ABB RAPID module: 0016EFE6

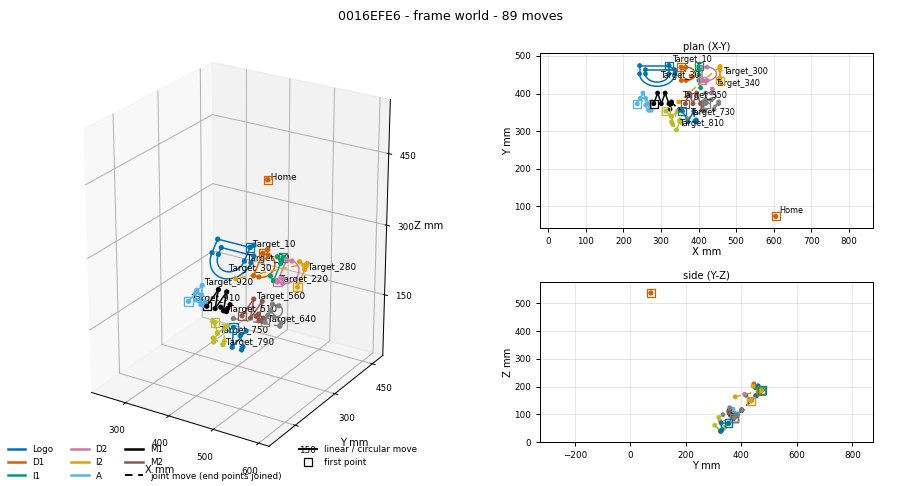
[picture p0: tool path of 0016EFE6 in frame world, 89 of 89 moves have a stored position in this frame; points joined in program order, loops and branches not executed]
MODULE Module1
    CONST robtarget Target_360:=[[614.368006487,-305.026841829,-535.49276156],[0.482962895,-0.129409515,-0.299950184,0.812422247],[-1,0,0,0],[9E+09,9E+09,9E+09,9E+09,9E+09,9E+09]];
    CONST robtarget Target_370:=[[614.368006487,-305.026841829,-535.49276156],[0.482962895,-0.129409515,-0.299950184,0.812422247],[-1,0,0,0],[9E+09,9E+09,9E+09,9E+09,9E+09,9E+09]];
    CONST robtarget Target_380:=[[614.368006487,-305.026841829,-535.49276156],[0.482962895,-0.129409515,-0.299950184,0.812422247],[-1,0,0,0],[9E+09,9E+09,9E+09,9E+09,9E+09,9E+09]];
    CONST robtarget Target_410:=[[614.368006487,-305.026841829,-535.49276156],[0.482962895,-0.129409515,-0.299950184,0.812422247],[-1,0,0,0],[9E+09,9E+09,9E+09,9E+09,9E+09,9E+09]];
    CONST robtarget Target_390:=[[614.368006487,-305.026841829,-535.49276156],[0.482962895,-0.129409515,-0.299950184,0.812422247],[-1,0,0,0],[9E+09,9E+09,9E+09,9E+09,9E+09,9E+09]];
    CONST robtarget Target_400:=[[614.368006487,-305.026841829,-535.49276156],[0.482962895,-0.129409515,-0.299950184,0.812422247],[-1,0,0,0],[9E+09,9E+09,9E+09,9E+09,9E+09,9E+09]];
    CONST robtarget Target_420:=[[614.368006487,-305.026841829,-535.49276156],[0.482962895,-0.129409515,-0.299950184,0.812422247],[-1,0,0,0],[9E+09,9E+09,9E+09,9E+09,9E+09,9E+09]];
    CONST robtarget Target_430:=[[614.368006487,-305.026841829,-535.49276156],[0.482962895,-0.129409515,-0.299950184,0.812422247],[-1,0,0,0],[9E+09,9E+09,9E+09,9E+09,9E+09,9E+09]];
    CONST robtarget Target_440:=[[614.368006487,-305.026841829,-535.49276156],[0.482962895,-0.129409515,-0.299950184,0.812422247],[-1,0,0,0],[9E+09,9E+09,9E+09,9E+09,9E+09,9E+09]];
    CONST robtarget Target_450:=[[614.368006487,-305.026841829,-535.49276156],[0.482962895,-0.129409515,-0.299950184,0.812422247],[-1,0,0,0],[9E+09,9E+09,9E+09,9E+09,9E+09,9E+09]];
    CONST robtarget Target_550:=[[186.614,135,0],[1,0,0,0],[0,0,0,0],[9E+09,9E+09,9E+09,9E+09,9E+09,9E+09]];
    CONST robtarget Target_560:=[[146.614,125,0],[1,0,0,0],[0,-2,1,0],[9E+09,9E+09,9E+09,9E+09,9E+09,9E+09]];
    CONST robtarget Target_570:=[[186.614,115,0],[1,0,0,0],[0,-2,1,0],[9E+09,9E+09,9E+09,9E+09,9E+09,9E+09]];
    CONST robtarget Target_580:=[[146.614,105,0],[1,0,0,0],[0,-2,1,0],[9E+09,9E+09,9E+09,9E+09,9E+09,9E+09]];
    CONST robtarget Target_590:=[[186.614,95,0],[1,0,0,0],[0,-2,1,0],[9E+09,9E+09,9E+09,9E+09,9E+09,9E+09]];
    CONST robtarget Target_620:=[[186.614143087,91.364778393,-24.569544894],[1,-0.00000011,0.000000243,0.000000801],[0,-2,1,0],[9E+09,9E+09,9E+09,9E+09,9E+09,9E+09]];
    CONST robtarget Target_600:=[[186.614,88,0],[1,0,0,0],[0,-2,1,0],[9E+09,9E+09,9E+09,9E+09,9E+09,9E+09]];
    CONST robtarget Target_610:=[[179.614,88,0],[1,0,0,0],[0,-2,1,0],[9E+09,9E+09,9E+09,9E+09,9E+09,9E+09]];
    CONST robtarget Target_630:=[[182.856287812,84.770817951,-30.544070021],[1,0.000000024,0.000000045,0.000000006],[0,-2,1,0],[9E+09,9E+09,9E+09,9E+09,9E+09,9E+09]];
    CONST robtarget Target_10:=[[43.067,178.883,0],[1,0,0,0],[0,-2,1,0],[9E+09,9E+09,9E+09,9E+09,9E+09,9E+09]];
    CONST robtarget Target_20:=[[74.267,178.883,0],[1,0,0,0],[0,-2,1,0],[9E+09,9E+09,9E+09,9E+09,9E+09,9E+09]];
    CONST robtarget Target_30:=[[105.467,210.083,0],[1,0,0,0],[0,-2,1,0],[9E+09,9E+09,9E+09,9E+09,9E+09,9E+09]];
    CONST robtarget Target_40:=[[74.267,241.283,0],[1,0,0,0],[0,-2,0,0],[9E+09,9E+09,9E+09,9E+09,9E+09,9E+09]];
    CONST robtarget Target_50:=[[58.667,241.283,0],[1,0,0,0],[0,-2,0,0],[9E+09,9E+09,9E+09,9E+09,9E+09,9E+09]];
    CONST robtarget Target_60:=[[58.667,163.283,0],[1,0,0,0],[0,-2,1,0],[9E+09,9E+09,9E+09,9E+09,9E+09,9E+09]];
    CONST robtarget Target_70:=[[74.267,163.283,0],[1,0,0,0],[0,-2,1,0],[9E+09,9E+09,9E+09,9E+09,9E+09,9E+09]];
    CONST robtarget Target_80:=[[121.067,210.083,0],[1,0,0,0],[0,-2,1,0],[9E+09,9E+09,9E+09,9E+09,9E+09,9E+09]];
    CONST robtarget Target_90:=[[74.267,256.883,0],[1,0,0,0],[0,-2,0,0],[9E+09,9E+09,9E+09,9E+09,9E+09,9E+09]];
    CONST robtarget Target_100:=[[43.067,256.883,0],[1,0,0,0],[0,-2,0,0],[9E+09,9E+09,9E+09,9E+09,9E+09,9E+09]];
    CONST robtarget Target_310:=[[43.067061989,160.806085243,-20.298551342],[1,-0.00000004,0.000000028,-0.000000016],[0,-2,1,0],[9E+09,9E+09,9E+09,9E+09,9E+09,9E+09]];
    CONST robtarget Target_110:=[[49.307,146.077,0],[1,0,0,0],[0,-2,1,0],[9E+09,9E+09,9E+09,9E+09,9E+09,9E+09]];
    CONST robtarget Target_120:=[[99.226985269,146.076975233,0.000011329],[1,0.000000004,0.00000003,-0.000000033],[0,-2,1,0],[9E+09,9E+09,9E+09,9E+09,9E+09,9E+09]];
    CONST robtarget Target_130:=[[99.227,133.597,0],[1,0,0,0],[0,-2,1,0],[9E+09,9E+09,9E+09,9E+09,9E+09,9E+09]];
    CONST robtarget Target_140:=[[74.267,108.637,0],[1,0,0,0],[0,-2,1,0],[9E+09,9E+09,9E+09,9E+09,9E+09,9E+09]];
    CONST robtarget Target_150:=[[49.307,133.597,0],[1,0,0,0],[0,-2,1,0],[9E+09,9E+09,9E+09,9E+09,9E+09,9E+09]];
    CONST robtarget Target_320:=[[49.307045531,119.232886712,-35.733129909],[1,-0.000000046,0.000000065,-0.00000006],[0,-2,1,0],[9E+09,9E+09,9E+09,9E+09,9E+09,9E+09]];
    CONST robtarget Target_160:=[[46.187,99.277,0],[1,0,0,0],[0,0,0,0],[9E+09,9E+09,9E+09,9E+09,9E+09,9E+09]];
    CONST robtarget Target_170:=[[52.427,99.277,0],[1,0,0,0],[0,-2,1,0],[9E+09,9E+09,9E+09,9E+09,9E+09,9E+09]];
    CONST robtarget Target_200:=[[55.43480685,99.276989953,-23.383322605],[1,-0.000000033,0.000000018,-0.000000049],[0,-2,1,0],[9E+09,9E+09,9E+09,9E+09,9E+09,9E+09]];
    CONST robtarget Target_180:=[[60.227,99.277,0],[1,0,0,0],[0,-2,1,0],[9E+09,9E+09,9E+09,9E+09,9E+09,9E+09]];
    CONST robtarget Target_190:=[[99.227,99.277,0],[1,0,0,0],[0,-2,1,0],[9E+09,9E+09,9E+09,9E+09,9E+09,9E+09]];
    CONST robtarget Target_330:=[[99.22721957,94.540167057,-27.618833902],[1,-0.000000004,0.00000006,-0.000000007],[0,-2,1,0],[9E+09,9E+09,9E+09,9E+09,9E+09,9E+09]];
    CONST robtarget Target_220:=[[99.227,89.917,0],[1,0,0,0],[0,-2,1,0],[9E+09,9E+09,9E+09,9E+09,9E+09,9E+09]];
    CONST robtarget Target_230:=[[99.227,77.437,0],[1,0,0,0],[0,-2,1,0],[9E+09,9E+09,9E+09,9E+09,9E+09,9E+09]];
    CONST robtarget Target_240:=[[74.267,52.477,0],[1,0,0,0],[0,-2,1,0],[9E+09,9E+09,9E+09,9E+09,9E+09,9E+09]];
    CONST robtarget Target_250:=[[49.307,77.437,0],[1,0,0,0],[0,-2,1,0],[9E+09,9E+09,9E+09,9E+09,9E+09,9E+09]];
    CONST robtarget Target_210:=[[49.307,89.917,0],[1,0,0,0],[0,-2,1,0],[9E+09,9E+09,9E+09,9E+09,9E+09,9E+09]];
    CONST robtarget Target_340:=[[99.227234287,63.232614277,-33.127627179],[1,-0.000000078,0.000000016,-0.000000084],[0,-2,1,0],[9E+09,9E+09,9E+09,9E+09,9E+09,9E+09]];
    CONST robtarget Target_290:=[[99.227,43.117,0],[1,0,0,0],[0,-2,1,0],[9E+09,9E+09,9E+09,9E+09,9E+09,9E+09]];
    CONST robtarget Target_280:=[[60.227,43.117,0],[1,0,0,0],[0,-2,1,0],[9E+09,9E+09,9E+09,9E+09,9E+09,9E+09]];
    CONST robtarget Target_300:=[[56.841349449,43.116999563,-32.2270308],[1,-0.000000054,0.000000041,0.000000045],[0,-2,1,0],[9E+09,9E+09,9E+09,9E+09,9E+09,9E+09]];
    CONST robtarget Target_270:=[[52.427,43.117,0],[1,0,0,0],[0,-2,1,0],[9E+09,9E+09,9E+09,9E+09,9E+09,9E+09]];
    CONST robtarget Target_260:=[[46.187,43.117,0],[1,0,0,0],[0,-2,1,0],[9E+09,9E+09,9E+09,9E+09,9E+09,9E+09]];
    CONST robtarget Target_350:=[[129.667098448,152.744988992,-50.230821834],[1,-0.000000071,0.000000063,0.000000069],[0,-2,1,0],[9E+09,9E+09,9E+09,9E+09,9E+09,9E+09]];
    CONST robtarget Target_460:=[[186.614,219,0],[1,0,0,0],[0,0,0,0],[9E+09,9E+09,9E+09,9E+09,9E+09,9E+09]];
    CONST robtarget Target_470:=[[146.614,209,0],[1,0,0,0],[0,-2,1,0],[9E+09,9E+09,9E+09,9E+09,9E+09,9E+09]];
    CONST robtarget Target_480:=[[186.614,199,0],[1,0,0,0],[0,-2,1,0],[9E+09,9E+09,9E+09,9E+09,9E+09,9E+09]];
    CONST robtarget Target_490:=[[146.614,189,0],[1,0,0,0],[0,-2,1,0],[9E+09,9E+09,9E+09,9E+09,9E+09,9E+09]];
    CONST robtarget Target_500:=[[186.614,179,0],[1,0,0,0],[0,-2,1,0],[9E+09,9E+09,9E+09,9E+09,9E+09,9E+09]];
    CONST robtarget Target_530:=[[186.614130113,175.925883793,-20.905174154],[1,-0.000000022,0.000000055,-0.000000082],[0,-2,1,0],[9E+09,9E+09,9E+09,9E+09,9E+09,9E+09]];
    CONST robtarget Target_510:=[[186.614,172,0],[1,0,0,0],[0,-2,1,0],[9E+09,9E+09,9E+09,9E+09,9E+09,9E+09]];
    CONST robtarget Target_520:=[[179.614,172,0],[1,0,0,0],[0,-2,1,0],[9E+09,9E+09,9E+09,9E+09,9E+09,9E+09]];
    CONST robtarget Target_540:=[[179.614118669,152.268392062,-31.694765884],[1,-0.000000012,0.000000036,0.000000018],[0,-2,1,0],[9E+09,9E+09,9E+09,9E+09,9E+09,9E+09]];
    CONST robtarget Target_640:=[[186.614,81,0],[1,0,0,0],[0,0,0,0],[9E+09,9E+09,9E+09,9E+09,9E+09,9E+09]];
    CONST robtarget Target_650:=[[146.614,81,0],[1,0,0,0],[0,-2,1,0],[9E+09,9E+09,9E+09,9E+09,9E+09,9E+09]];
    CONST robtarget Target_660:=[[146.614,66,0],[1,0,0,0],[0,-2,1,0],[9E+09,9E+09,9E+09,9E+09,9E+09,9E+09]];
    CONST robtarget Target_670:=[[159.114,53.5,0],[1,0,0,0],[0,-2,1,0],[9E+09,9E+09,9E+09,9E+09,9E+09,9E+09]];
    CONST robtarget Target_680:=[[171.614,66,0],[1,0,0,0],[0,-2,1,0],[9E+09,9E+09,9E+09,9E+09,9E+09,9E+09]];
    CONST robtarget Target_690:=[[171.614,81,0],[1,0,0,0],[0,-2,1,0],[9E+09,9E+09,9E+09,9E+09,9E+09,9E+09]];
    CONST robtarget Target_720:=[[171.614154806,58.991203706,-36.638059024],[1,-0.000000034,0.000000051,-0.000000007],[0,-2,1,0],[9E+09,9E+09,9E+09,9E+09,9E+09,9E+09]];
    CONST robtarget Target_700:=[[179.614,46.5,0],[1,0,0,0],[0,-2,1,0],[9E+09,9E+09,9E+09,9E+09,9E+09,9E+09]];
    CONST robtarget Target_710:=[[186.614,46.5,0],[1,0,0,0],[0,-2,1,0],[9E+09,9E+09,9E+09,9E+09,9E+09,9E+09]];
    CONST robtarget Target_730:=[[206.575839686,130.575385522,-36.062606272],[1,-0.000000061,0.000000016,-0.000000213],[0,-2,1,0],[9E+09,9E+09,9E+09,9E+09,9E+09,9E+09]];
    CONST robtarget Target_740:=[[214.649,187,0],[1,0,0,0],[0,0,0,0],[9E+09,9E+09,9E+09,9E+09,9E+09,9E+09]];
    CONST robtarget Target_750:=[[234.649,172,0],[1,0,0,0],[0,-2,1,0],[9E+09,9E+09,9E+09,9E+09,9E+09,9E+09]];
    CONST robtarget Target_760:=[[214.649,157,0],[1,0,0,0],[0,-2,1,0],[9E+09,9E+09,9E+09,9E+09,9E+09,9E+09]];
    CONST robtarget Target_800:=[[224.454054793,169.052592344,-39.983761207],[1,-0.000000024,0.000000053,-0.000000097],[0,-2,1,0],[9E+09,9E+09,9E+09,9E+09,9E+09,9E+09]];
    CONST robtarget Target_770:=[[254.649,172,0],[1,0,0,0],[0,-2,1,0],[9E+09,9E+09,9E+09,9E+09,9E+09,9E+09]];
    CONST robtarget Target_810:=[[254.649337072,159.007769138,-30.298077251],[1,-0.000000027,0.000000051,-0.000000098],[0,-2,1,0],[9E+09,9E+09,9E+09,9E+09,9E+09,9E+09]];
    CONST robtarget Target_790:=[[254.649,150,0],[1,0,0,0],[0,-2,1,0],[9E+09,9E+09,9E+09,9E+09,9E+09,9E+09]];
    CONST robtarget Target_780:=[[247.649,150,0],[1,0,0,0],[0,-2,1,0],[9E+09,9E+09,9E+09,9E+09,9E+09,9E+09]];
    CONST robtarget Target_820:=[[229.743211704,145.004792269,-27.634877565],[1,-0.000000014,0.000000023,0.000000082],[0,-2,1,0],[9E+09,9E+09,9E+09,9E+09,9E+09,9E+09]];
    CONST robtarget Target_830:=[[214.649,143,0],[1,0,0,0],[0,0,0,0],[9E+09,9E+09,9E+09,9E+09,9E+09,9E+09]];
    CONST robtarget Target_840:=[[254.649,128,0],[1,0,0,0],[0,-2,1,0],[9E+09,9E+09,9E+09,9E+09,9E+09,9E+09]];
    CONST robtarget Target_850:=[[214.649,113,0],[1,0,0,0],[0,-2,1,0],[9E+09,9E+09,9E+09,9E+09,9E+09,9E+09]];
    CONST robtarget Target_880:=[[232.237809143,110.203682172,-19.826551886],[1,-0.000000178,0.000000032,0.000000095],[0,-2,1,0],[9E+09,9E+09,9E+09,9E+09,9E+09,9E+09]];
    CONST robtarget Target_860:=[[247.649,106,0],[1,0,0,0],[0,-2,1,0],[9E+09,9E+09,9E+09,9E+09,9E+09,9E+09]];
    CONST robtarget Target_870:=[[254.649,106,0],[1,0,0,0],[0,-2,1,0],[9E+09,9E+09,9E+09,9E+09,9E+09,9E+09]];
    CONST robtarget Home:=[[605.026172128,73.5,537.625162051],[0.500000001,0,0.866025403,0],[-1,0,-1,0],[9E+09,9E+09,9E+09,9E+09,9E+09,9E+09]];
    TASK PERS wobjdata Workobject_1:=[FALSE,TRUE,"",[[500,512.132,212.132],[0.27059805,-0.653281482,0.653281482,0.27059805]],[[0,0,-10],[1,0,0,0]]];
    CONST robtarget Target_900:=[[614.368006487,-305.026841829,-535.49276156],[0.482962895,-0.129409515,-0.299950184,0.812422247],[-1,0,0,0],[9E+09,9E+09,9E+09,9E+09,9E+09,9E+09]];
    CONST robtarget Target_910:=[[186.613,263,0],[1,0,0,0],[0,0,0,0],[9E+09,9E+09,9E+09,9E+09,9E+09,9E+09]];
    CONST robtarget Target_920:=[[146.613,248,0],[1,0,0,0],[0,0,-1,0],[9E+09,9E+09,9E+09,9E+09,9E+09,9E+09]];
    CONST robtarget Target_930:=[[186.613,233,0],[1,0,0,0],[0,0,-1,0],[9E+09,9E+09,9E+09,9E+09,9E+09,9E+09]];
    CONST robtarget Target_930_4:=[[186.613,233,-25],[1,0,0,0],[0,0,-1,0],[9E+09,9E+09,9E+09,9E+09,9E+09,9E+09]];
    CONST robtarget Target_940:=[[166.613,255.5,0],[1,0,0,0],[0,0,-1,0],[9E+09,9E+09,9E+09,9E+09,9E+09,9E+09]];
    CONST robtarget Target_950:=[[166.613,240.5,0],[1,0,0,0],[0,0,-1,0],[9E+09,9E+09,9E+09,9E+09,9E+09,9E+09]];
    CONST robtarget Target_950_2:=[[166.613,240.5,-25],[1,0,0,0],[0,0,-1,0],[9E+09,9E+09,9E+09,9E+09,9E+09,9E+09]];
    CONST robtarget Target_970:=[[179.613,226,0],[1,0,0,0],[0,0,-1,0],[9E+09,9E+09,9E+09,9E+09,9E+09,9E+09]];
    CONST robtarget Target_960:=[[186.613,226,0],[1,0,0,0],[0,0,-1,0],[9E+09,9E+09,9E+09,9E+09,9E+09,9E+09]];
    CONST robtarget Target_960_2:=[[186.613,226,-25],[1,0,0,0],[0,0,-1,0],[9E+09,9E+09,9E+09,9E+09,9E+09,9E+09]];
    PERS tooldata MyNewTool:=[TRUE,[[73.5,-73.5,156.444],[1,0,0,0]],[1,[0,0,1],[1,0,0,0],0,0,0]];
    PROC Logo()
        MoveJ Target_10,v300,fine,MyNewTool\WObj:=Workobject_1;
        MoveL Target_20,v100,fine,MyNewTool\WObj:=Workobject_1;
        MoveC Target_30,Target_40,v100,fine,MyNewTool\WObj:=Workobject_1;
        MoveL Target_50,v100,fine,MyNewTool\WObj:=Workobject_1;
        MoveL Target_60,v100,fine,MyNewTool\WObj:=Workobject_1;
        MoveL Target_70,v100,fine,MyNewTool\WObj:=Workobject_1;
        MoveC Target_80,Target_90,v100,fine,MyNewTool\WObj:=Workobject_1;
        MoveL Target_100,v100,fine,MyNewTool\WObj:=Workobject_1;
        MoveL Target_10,v100,fine,MyNewTool\WObj:=Workobject_1;
        MoveJ Target_310,v300,z10,MyNewTool\WObj:=Workobject_1;

    ENDPROC
    PROC D1()
        MoveJ Target_110,v300,fine,MyNewTool\WObj:=Workobject_1;
        MoveL Target_120,v100,fine,MyNewTool\WObj:=Workobject_1;
        MoveL Target_130,v100,fine,MyNewTool\WObj:=Workobject_1;
        MoveC Target_140,Target_150,v100,fine,MyNewTool\WObj:=Workobject_1;
        MoveL Target_110,v100,fine,MyNewTool\WObj:=Workobject_1;
        MoveJ Target_320,v300,z10,MyNewTool\WObj:=Workobject_1;

    ENDPROC
    PROC I1()
        MoveJ Target_160,v300,fine,MyNewTool\WObj:=Workobject_1;
        MoveL Target_170,v100,fine,MyNewTool\WObj:=Workobject_1;
        MoveJ Target_200,v300,z10,MyNewTool\WObj:=Workobject_1;
        MoveJ Target_180,v300,fine,MyNewTool\WObj:=Workobject_1;
        MoveL Target_190,v100,fine,MyNewTool\WObj:=Workobject_1;
        MoveJ Target_330,v300,z10,MyNewTool\WObj:=Workobject_1;

    ENDPROC
    PROC D2()
        MoveJ Target_220,v300,fine,MyNewTool\WObj:=Workobject_1;
        MoveL Target_230,v100,fine,MyNewTool\WObj:=Workobject_1;
        MoveC Target_240,Target_250,v100,fine,MyNewTool\WObj:=Workobject_1;
        MoveL Target_210,v100,fine,MyNewTool\WObj:=Workobject_1;
        MoveL Target_220,v100,fine,MyNewTool\WObj:=Workobject_1;
        MoveJ Target_340,v300,z10,MyNewTool\WObj:=Workobject_1;

    ENDPROC
    PROC I2()
        MoveJ Target_290,v300,fine,MyNewTool\WObj:=Workobject_1;
        MoveL Target_280,v100,fine,MyNewTool\WObj:=Workobject_1;
        MoveJ Target_300,v300,z10,MyNewTool\WObj:=Workobject_1;
        MoveJ Target_270,v300,fine,MyNewTool\WObj:=Workobject_1;
        MoveL Target_260,v100,fine,MyNewTool\WObj:=Workobject_1;
        MoveJ Target_350,v300,z10,MyNewTool\WObj:=Workobject_1;

    ENDPROC
    PROC A()
        MoveJ Target_910,v300,fine,MyNewTool\WObj:=Workobject_1;
        MoveL Target_920,v100,fine,MyNewTool\WObj:=Workobject_1;
        MoveL Target_930,v100,fine,MyNewTool\WObj:=Workobject_1;
        MoveJ Target_930_4,v300,z10,MyNewTool\WObj:=Workobject_1;
        MoveJ Target_940,v300,fine,MyNewTool\WObj:=Workobject_1;
        MoveL Target_950,v100,fine,MyNewTool\WObj:=Workobject_1;
        MoveJ Target_950_2,v300,z10,MyNewTool\WObj:=Workobject_1;
        MoveJ Target_970,v300,fine,MyNewTool\WObj:=Workobject_1;
        MoveL Target_960,v100,fine,MyNewTool\WObj:=Workobject_1;
        MoveJ Target_960_2,v300,z10,MyNewTool\WObj:=Workobject_1;
    ENDPROC
    PROC M1()
        MoveJ Target_460,v300,fine,MyNewTool\WObj:=Workobject_1;
        MoveL Target_470,v100,fine,MyNewTool\WObj:=Workobject_1;
        MoveL Target_480,v100,fine,MyNewTool\WObj:=Workobject_1;
        MoveL Target_490,v100,fine,MyNewTool\WObj:=Workobject_1;
        MoveL Target_500,v100,fine,MyNewTool\WObj:=Workobject_1;
        MoveJ Target_530,v300,z10,MyNewTool\WObj:=Workobject_1;
        MoveJ Target_510,v300,fine,MyNewTool\WObj:=Workobject_1;
        MoveL Target_520,v100,fine,MyNewTool\WObj:=Workobject_1;
        MoveJ Target_540,v300,z10,MyNewTool\WObj:=Workobject_1;

    ENDPROC
    PROC M2()
        MoveJ Target_550,v300,fine,MyNewTool\WObj:=Workobject_1;
        MoveL Target_560,v100,fine,MyNewTool\WObj:=Workobject_1;
        MoveL Target_570,v100,fine,MyNewTool\WObj:=Workobject_1;
        MoveL Target_580,v100,fine,MyNewTool\WObj:=Workobject_1;
        MoveL Target_590,v100,fine,MyNewTool\WObj:=Workobject_1;
        MoveJ Target_620,v300,z10,MyNewTool\WObj:=Workobject_1;
        MoveJ Target_600,v300,fine,MyNewTool\WObj:=Workobject_1;
        MoveL Target_610,v100,fine,MyNewTool\WObj:=Workobject_1;
        MoveJ Target_630,v300,z10,MyNewTool\WObj:=Workobject_1;

    ENDPROC
    PROC P()
        MoveJ Target_640,v300,fine,MyNewTool\WObj:=Workobject_1;
        MoveL Target_650,v100,fine,MyNewTool\WObj:=Workobject_1;
        MoveL Target_660,v100,fine,MyNewTool\WObj:=Workobject_1;
        MoveC Target_670,Target_680,v100,fine,MyNewTool\WObj:=Workobject_1;
        MoveL Target_690,v100,fine,MyNewTool\WObj:=Workobject_1;
        MoveJ Target_720,v300,z10,MyNewTool\WObj:=Workobject_1;
        MoveJ Target_700,v300,fine,MyNewTool\WObj:=Workobject_1;
        MoveL Target_710,v100,fine,MyNewTool\WObj:=Workobject_1;
        MoveJ Target_730,v300,z10,MyNewTool\WObj:=Workobject_1;

    ENDPROC
    PROC Y()
        MoveJ Target_740,v300,fine,MyNewTool\WObj:=Workobject_1;
        MoveL Target_750,v100,fine,MyNewTool\WObj:=Workobject_1;
        MoveL Target_760,v100,fine,MyNewTool\WObj:=Workobject_1;
        MoveJ Target_800,v300,z10,MyNewTool\WObj:=Workobject_1;
        MoveJ Target_750,v300,fine,MyNewTool\WObj:=Workobject_1;
        MoveL Target_770,v100,fine,MyNewTool\WObj:=Workobject_1;
        MoveJ Target_810,v300,z10,MyNewTool\WObj:=Workobject_1;
        MoveJ Target_790,v300,fine,MyNewTool\WObj:=Workobject_1;
        MoveL Target_780,v100,fine,MyNewTool\WObj:=Workobject_1;
        MoveJ Target_820,v300,z10,MyNewTool\WObj:=Workobject_1;

    ENDPROC
    PROC V()
        MoveJ Target_830,v300,fine,MyNewTool\WObj:=Workobject_1;
        MoveL Target_840,v100,fine,MyNewTool\WObj:=Workobject_1;
        MoveL Target_850,v100,fine,MyNewTool\WObj:=Workobject_1;
        MoveJ Target_880,v300,z10,MyNewTool\WObj:=Workobject_1;
        MoveJ Target_860,v300,fine,MyNewTool\WObj:=Workobject_1;
        MoveL Target_870,v100,fine,MyNewTool\WObj:=Workobject_1;

    ENDPROC
    PROC Main()
        MoveJ Home,v300,z10,MyNewTool\WObj:=wobj0;
        Logo;
        D1;
        I1;
        D2;
        I2;
        A;
        M1;
        M2;
        P;
        Y;
        V;
        MoveJ Home,v300,z10,MyNewTool\WObj:=wobj0;
    ENDPROC
ENDMODULE
